// TIA Portal V20 export
FUNCTION "06 T5 EXCENTRIC Output" : Void   // FC1618, LAD
TITLE = OUTPUT
{ S7_Optimized_Access := 'TRUE' }
// stored: AutoNumber false, SetENOAutomatically false
   VAR_TEMP
      Aux_real : Real;
      Aux_dint : DInt;
      Aux_uint : UInt;
      Aux_Bool : Bool;
      Aux_OS : Bool;
   END_VAR
   VAR_TEMP   // added for the SCL form of the ladder/FBD networks
      _w1 : Bool;
      _w2 : Bool;
   END_VAR
BEGIN

REGION Network 1: ============= INTERLOCKS MOVING FORWARD =============
END_REGION

REGION Network 2: Interlocks Move FORWARD - Permanent Conditions
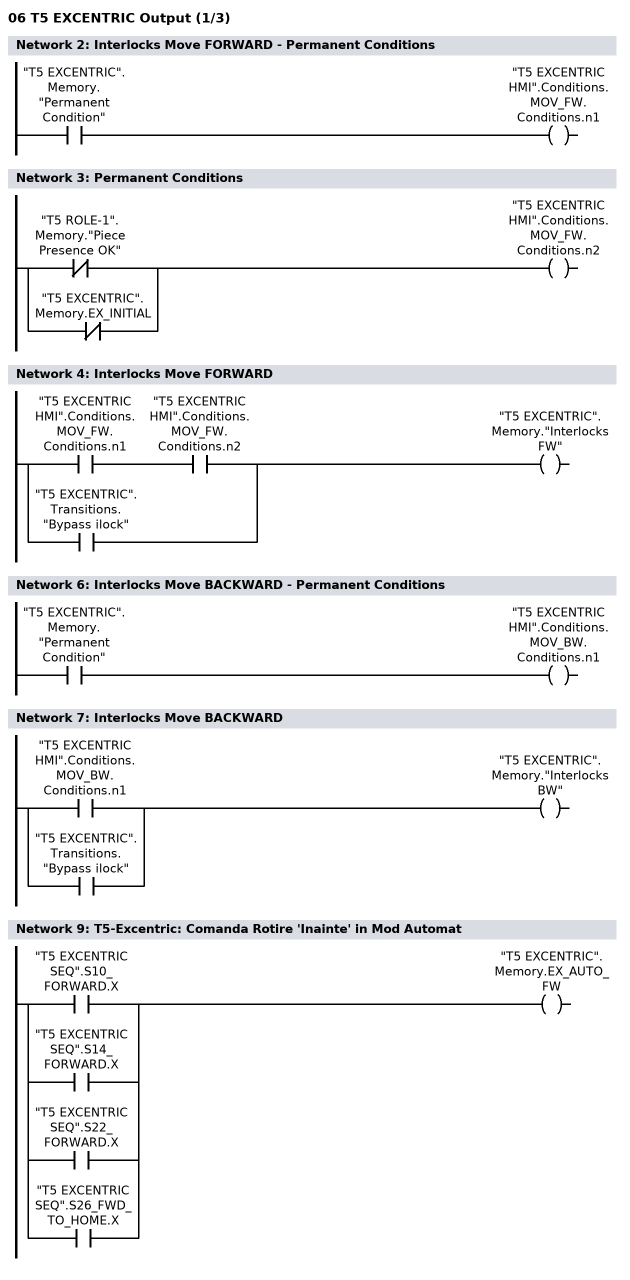
   RUNG wire#powerrail
      Contact( "T5 EXCENTRIC".Memory."Permanent Condition" )
      Coil( "T5 EXCENTRIC HMI".Conditions.MOV_FW.Conditions.n1 )
   END_RUNG
   // the same network as SCL:
   "T5 EXCENTRIC HMI".Conditions.MOV_FW.Conditions.n1 := "T5 EXCENTRIC".Memory."Permanent Condition";
END_REGION

REGION Network 3: Permanent Conditions
   RUNG wire#powerrail
      I_Contact( "T5 ROLE-1".Memory."Piece Presence OK" )
      wire#w1
      Coil( "T5 EXCENTRIC HMI".Conditions.MOV_FW.Conditions.n2 )
   END_RUNG
   RUNG wire#powerrail
      I_Contact( "T5 EXCENTRIC".Memory.EX_INITIAL )
   END_RUNG wire#w1
   // the same network as SCL:
   "T5 EXCENTRIC HMI".Conditions.MOV_FW.Conditions.n2 := NOT "T5 ROLE-1".Memory."Piece Presence OK" OR NOT "T5 EXCENTRIC".Memory.EX_INITIAL;
END_REGION

REGION Network 4: Interlocks Move FORWARD
   RUNG wire#powerrail
      Contact( "T5 EXCENTRIC HMI".Conditions.MOV_FW.Conditions.n1 )
      Contact( "T5 EXCENTRIC HMI".Conditions.MOV_FW.Conditions.n2 )
      wire#w1
      Coil( "T5 EXCENTRIC".Memory."Interlocks FW" )
   END_RUNG
   RUNG wire#powerrail
      Contact( "T5 EXCENTRIC".Transitions."Bypass ilock" )
   END_RUNG wire#w1
   // the same network as SCL:
   "T5 EXCENTRIC".Memory."Interlocks FW" := ("T5 EXCENTRIC HMI".Conditions.MOV_FW.Conditions.n1 AND "T5 EXCENTRIC HMI".Conditions.MOV_FW.Conditions.n2) OR "T5 EXCENTRIC".Transitions."Bypass ilock";
END_REGION

REGION Network 5: ============= INTERLOCKS MOVING BACKWARD =============
END_REGION

REGION Network 6: Interlocks Move BACKWARD - Permanent Conditions
   RUNG wire#powerrail
      Contact( "T5 EXCENTRIC".Memory."Permanent Condition" )
      Coil( "T5 EXCENTRIC HMI".Conditions.MOV_BW.Conditions.n1 )
   END_RUNG
   // the same network as SCL:
   "T5 EXCENTRIC HMI".Conditions.MOV_BW.Conditions.n1 := "T5 EXCENTRIC".Memory."Permanent Condition";
END_REGION

REGION Network 7: Interlocks Move BACKWARD
   RUNG wire#powerrail
      Contact( "T5 EXCENTRIC HMI".Conditions.MOV_BW.Conditions.n1 )
      wire#w1
      Coil( "T5 EXCENTRIC".Memory."Interlocks BW" )
   END_RUNG
   RUNG wire#powerrail
      Contact( "T5 EXCENTRIC".Transitions."Bypass ilock" )
   END_RUNG wire#w1
   // the same network as SCL:
   "T5 EXCENTRIC".Memory."Interlocks BW" := "T5 EXCENTRIC HMI".Conditions.MOV_BW.Conditions.n1 OR "T5 EXCENTRIC".Transitions."Bypass ilock";
END_REGION

REGION Network 8: ============ COMMANDS ============
END_REGION

REGION Network 9: T5-Excentric: Comanda Rotire 'Inainte' in Mod Automat
   RUNG wire#powerrail
      Contact( "T5 EXCENTRIC SEQ".S10_FORWARD.X )
      wire#w1
      Coil( "T5 EXCENTRIC".Memory.EX_AUTO_FW )
   END_RUNG
   RUNG wire#powerrail
      Contact( "T5 EXCENTRIC SEQ".S14_FORWARD.X )
   END_RUNG wire#w1
   RUNG wire#powerrail
      Contact( "T5 EXCENTRIC SEQ".S22_FORWARD.X )
   END_RUNG wire#w1
   RUNG wire#powerrail
      Contact( "T5 EXCENTRIC SEQ".S26_FWD_TO_HOME.X )
   END_RUNG wire#w1
   // the same network as SCL:
   "T5 EXCENTRIC".Memory.EX_AUTO_FW := "T5 EXCENTRIC SEQ".S10_FORWARD.X OR "T5 EXCENTRIC SEQ".S14_FORWARD.X OR "T5 EXCENTRIC SEQ".S22_FORWARD.X OR "T5 EXCENTRIC SEQ".S26_FWD_TO_HOME.X;
END_REGION

REGION Network 10: T5-Excentric: Comanda Rotire 'Inainte' in Mod Manual
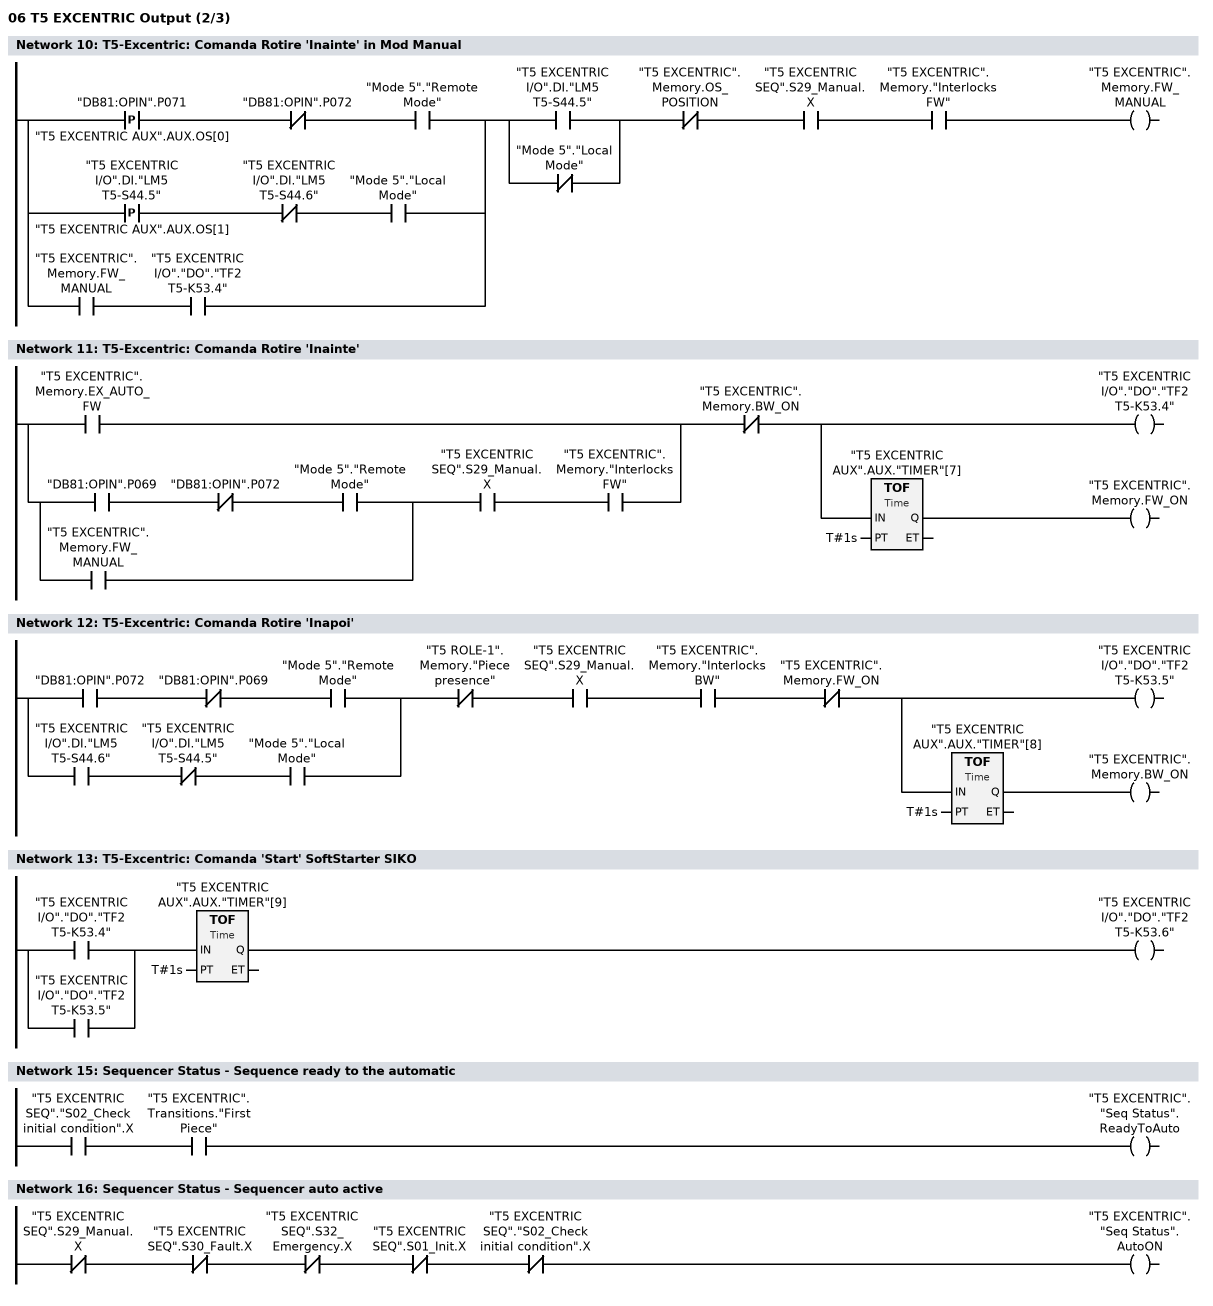
   RUNG wire#powerrail
      P_Contact(operand := "DB81:OPIN".P071, bit := "T5 EXCENTRIC AUX".AUX.OS[0])
      I_Contact( "DB81:OPIN".P072 )
      Contact( "Mode 5"."Remote Mode" )
      wire#w1
      Contact( "T5 EXCENTRIC I/O".DI."LM5 T5-S44.5" )
      wire#w2
      I_Contact( "T5 EXCENTRIC".Memory.OS_POSITION )
      Contact( "T5 EXCENTRIC SEQ".S29_Manual.X )
      Contact( "T5 EXCENTRIC".Memory."Interlocks FW" )
      Coil( "T5 EXCENTRIC".Memory.FW_MANUAL )
   END_RUNG
   RUNG wire#powerrail
      P_Contact(operand := "T5 EXCENTRIC I/O".DI."LM5 T5-S44.5", bit := "T5 EXCENTRIC AUX".AUX.OS[1])
      I_Contact( "T5 EXCENTRIC I/O".DI."LM5 T5-S44.6" )
      Contact( "Mode 5"."Local Mode" )
   END_RUNG wire#w1
   RUNG wire#powerrail
      Contact( "T5 EXCENTRIC".Memory.FW_MANUAL )
      Contact( "T5 EXCENTRIC I/O"."DO"."TF2 T5-K53.4" )
   END_RUNG wire#w1
   RUNG wire#w1
      I_Contact( "Mode 5"."Local Mode" )
   END_RUNG wire#w2
   // the same network as SCL:
   #_w1 := "DB81:OPIN".P071 AND NOT "T5 EXCENTRIC AUX".AUX.OS[0];   // rising edge of "DB81:OPIN".P071
   "T5 EXCENTRIC AUX".AUX.OS[0] := "DB81:OPIN".P071;
   #_w2 := "T5 EXCENTRIC I/O".DI."LM5 T5-S44.5" AND NOT "T5 EXCENTRIC AUX".AUX.OS[1];   // rising edge of "T5 EXCENTRIC I/O".DI."LM5 T5-S44.5"
   "T5 EXCENTRIC AUX".AUX.OS[1] := "T5 EXCENTRIC I/O".DI."LM5 T5-S44.5";
   "T5 EXCENTRIC".Memory.FW_MANUAL := ((#_w1 AND NOT "DB81:OPIN".P072 AND "Mode 5"."Remote Mode") OR (#_w2 AND NOT "T5 EXCENTRIC I/O".DI."LM5 T5-S44.6" AND "Mode 5"."Local Mode") OR ("T5 EXCENTRIC".Memory.FW_MANUAL AND "T5 EXCENTRIC I/O"."DO"."TF2 T5-K53.4")) AND ("T5 EXCENTRIC I/O".DI."LM5 T5-S44.5" OR NOT "Mode 5"."Local Mode") AND NOT "T5 EXCENTRIC".Memory.OS_POSITION AND "T5 EXCENTRIC SEQ".S29_Manual.X AND "T5 EXCENTRIC".Memory."Interlocks FW";
END_REGION

REGION Network 11: T5-Excentric: Comanda Rotire 'Inainte'
   RUNG wire#powerrail
      Contact( "T5 EXCENTRIC".Memory.EX_AUTO_FW )
      wire#w1
      I_Contact( "T5 EXCENTRIC".Memory.BW_ON )
      wire#w3
      Coil( "T5 EXCENTRIC I/O"."DO"."TF2 T5-K53.4" )
   END_RUNG
   RUNG wire#powerrail
      Contact( "DB81:OPIN".P069 )
      I_Contact( "DB81:OPIN".P072 )
      Contact( "Mode 5"."Remote Mode" )
      wire#w2
      Contact( "T5 EXCENTRIC SEQ".S29_Manual.X )
      Contact( "T5 EXCENTRIC".Memory."Interlocks FW" )
   END_RUNG wire#w1
   RUNG wire#powerrail
      Contact( "T5 EXCENTRIC".Memory.FW_MANUAL )
   END_RUNG wire#w2
   RUNG wire#w3
      { S7_Templates := "time_type := Time" } "T5 EXCENTRIC AUX".AUX."TIMER"[7].TOF(pt := T#1s, et =>)
      Coil( "T5 EXCENTRIC".Memory.FW_ON )
   END_RUNG
   // the same network as SCL:
   "T5 EXCENTRIC I/O"."DO"."TF2 T5-K53.4" := ("T5 EXCENTRIC".Memory.EX_AUTO_FW OR ((("DB81:OPIN".P069 AND NOT "DB81:OPIN".P072 AND "Mode 5"."Remote Mode") OR "T5 EXCENTRIC".Memory.FW_MANUAL) AND "T5 EXCENTRIC SEQ".S29_Manual.X AND "T5 EXCENTRIC".Memory."Interlocks FW")) AND NOT "T5 EXCENTRIC".Memory.BW_ON;
   "T5 EXCENTRIC AUX".AUX."TIMER"[7].TOF(IN := "T5 EXCENTRIC I/O"."DO"."TF2 T5-K53.4", PT := T#1s);
   "T5 EXCENTRIC".Memory.FW_ON := "T5 EXCENTRIC AUX".AUX."TIMER"[7].Q;
END_REGION

REGION Network 12: T5-Excentric: Comanda Rotire 'Inapoi'
   RUNG wire#powerrail
      Contact( "DB81:OPIN".P072 )
      I_Contact( "DB81:OPIN".P069 )
      Contact( "Mode 5"."Remote Mode" )
      wire#w1
      I_Contact( "T5 ROLE-1".Memory."Piece presence" )
      Contact( "T5 EXCENTRIC SEQ".S29_Manual.X )
      Contact( "T5 EXCENTRIC".Memory."Interlocks BW" )
      I_Contact( "T5 EXCENTRIC".Memory.FW_ON )
      wire#w2
      Coil( "T5 EXCENTRIC I/O"."DO"."TF2 T5-K53.5" )
   END_RUNG
   RUNG wire#powerrail
      Contact( "T5 EXCENTRIC I/O".DI."LM5 T5-S44.6" )
      I_Contact( "T5 EXCENTRIC I/O".DI."LM5 T5-S44.5" )
      Contact( "Mode 5"."Local Mode" )
   END_RUNG wire#w1
   RUNG wire#w2
      { S7_Templates := "time_type := Time" } "T5 EXCENTRIC AUX".AUX."TIMER"[8].TOF(pt := T#1s, et =>)
      Coil( "T5 EXCENTRIC".Memory.BW_ON )
   END_RUNG
   // the same network as SCL:
   "T5 EXCENTRIC I/O"."DO"."TF2 T5-K53.5" := (("DB81:OPIN".P072 AND NOT "DB81:OPIN".P069 AND "Mode 5"."Remote Mode") OR ("T5 EXCENTRIC I/O".DI."LM5 T5-S44.6" AND NOT "T5 EXCENTRIC I/O".DI."LM5 T5-S44.5" AND "Mode 5"."Local Mode")) AND NOT "T5 ROLE-1".Memory."Piece presence" AND "T5 EXCENTRIC SEQ".S29_Manual.X AND "T5 EXCENTRIC".Memory."Interlocks BW" AND NOT "T5 EXCENTRIC".Memory.FW_ON;
   "T5 EXCENTRIC AUX".AUX."TIMER"[8].TOF(IN := "T5 EXCENTRIC I/O"."DO"."TF2 T5-K53.5", PT := T#1s);
   "T5 EXCENTRIC".Memory.BW_ON := "T5 EXCENTRIC AUX".AUX."TIMER"[8].Q;
END_REGION

REGION Network 13: T5-Excentric: Comanda 'Start' SoftStarter SIKO
   RUNG wire#powerrail
      Contact( "T5 EXCENTRIC I/O"."DO"."TF2 T5-K53.4" )
      wire#w1
      { S7_Templates := "time_type := Time" } "T5 EXCENTRIC AUX".AUX."TIMER"[9].TOF(pt := T#1s, et =>)
      Coil( "T5 EXCENTRIC I/O"."DO"."TF2 T5-K53.6" )
   END_RUNG
   RUNG wire#powerrail
      Contact( "T5 EXCENTRIC I/O"."DO"."TF2 T5-K53.5" )
   END_RUNG wire#w1
   // the same network as SCL:
   "T5 EXCENTRIC AUX".AUX."TIMER"[9].TOF(IN := "T5 EXCENTRIC I/O"."DO"."TF2 T5-K53.4" OR "T5 EXCENTRIC I/O"."DO"."TF2 T5-K53.5",
                           PT := T#1s);
   "T5 EXCENTRIC I/O"."DO"."TF2 T5-K53.6" := "T5 EXCENTRIC AUX".AUX."TIMER"[9].Q;
END_REGION

REGION Network 14: ================== SEQUENCER STATUS ==================
END_REGION

REGION Network 15: Sequencer Status - Sequence ready to the automatic
   RUNG wire#powerrail
      Contact( "T5 EXCENTRIC SEQ"."S02_Check initial condition".X )
      Contact( "T5 EXCENTRIC".Transitions."First Piece" )
      Coil( "T5 EXCENTRIC"."Seq Status".ReadyToAuto )
   END_RUNG
   // the same network as SCL:
   "T5 EXCENTRIC"."Seq Status".ReadyToAuto := "T5 EXCENTRIC SEQ"."S02_Check initial condition".X AND "T5 EXCENTRIC".Transitions."First Piece";
END_REGION

REGION Network 16: Sequencer Status - Sequencer auto active
   RUNG wire#powerrail
      I_Contact( "T5 EXCENTRIC SEQ".S29_Manual.X )
      I_Contact( "T5 EXCENTRIC SEQ".S30_Fault.X )
      I_Contact( "T5 EXCENTRIC SEQ".S32_Emergency.X )
      I_Contact( "T5 EXCENTRIC SEQ".S01_Init.X )
      I_Contact( "T5 EXCENTRIC SEQ"."S02_Check initial condition".X )
      Coil( "T5 EXCENTRIC"."Seq Status".AutoON )
   END_RUNG
   // the same network as SCL:
   "T5 EXCENTRIC"."Seq Status".AutoON := NOT "T5 EXCENTRIC SEQ".S29_Manual.X AND NOT "T5 EXCENTRIC SEQ".S30_Fault.X AND NOT "T5 EXCENTRIC SEQ".S32_Emergency.X AND NOT "T5 EXCENTRIC SEQ".S01_Init.X AND NOT "T5 EXCENTRIC SEQ"."S02_Check initial condition".X;
END_REGION

REGION Network 17: Sequencer Status - Sequencer wait piece
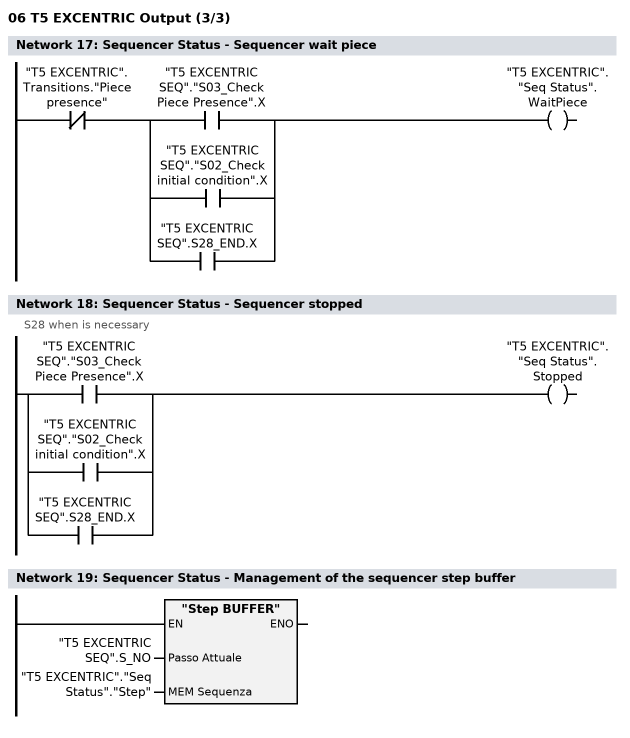
   RUNG wire#powerrail
      I_Contact( "T5 EXCENTRIC".Transitions."Piece presence" )
      wire#w1
      Contact( "T5 EXCENTRIC SEQ"."S03_Check Piece Presence".X )
      wire#w2
      Coil( "T5 EXCENTRIC"."Seq Status".WaitPiece )
   END_RUNG
   RUNG wire#w1
      Contact( "T5 EXCENTRIC SEQ"."S02_Check initial condition".X )
   END_RUNG wire#w2
   RUNG wire#w1
      Contact( "T5 EXCENTRIC SEQ".S28_END.X )
   END_RUNG wire#w2
   // the same network as SCL:
   "T5 EXCENTRIC"."Seq Status".WaitPiece := NOT "T5 EXCENTRIC".Transitions."Piece presence" AND ("T5 EXCENTRIC SEQ"."S03_Check Piece Presence".X OR "T5 EXCENTRIC SEQ"."S02_Check initial condition".X OR "T5 EXCENTRIC SEQ".S28_END.X);
END_REGION

REGION Network 18: Sequencer Status - Sequencer stopped
   // S28 when is necessary
   RUNG wire#powerrail
      Contact( "T5 EXCENTRIC SEQ"."S03_Check Piece Presence".X )
      wire#w1
      Coil( "T5 EXCENTRIC"."Seq Status".Stopped )
   END_RUNG
   RUNG wire#powerrail
      Contact( "T5 EXCENTRIC SEQ"."S02_Check initial condition".X )
   END_RUNG wire#w1
   RUNG wire#powerrail
      Contact( "T5 EXCENTRIC SEQ".S28_END.X )
   END_RUNG wire#w1
   // the same network as SCL:
   "T5 EXCENTRIC"."Seq Status".Stopped := "T5 EXCENTRIC SEQ"."S03_Check Piece Presence".X OR "T5 EXCENTRIC SEQ"."S02_Check initial condition".X OR "T5 EXCENTRIC SEQ".S28_END.X;
END_REGION

REGION Network 19: Sequencer Status - Management of the sequencer step buffer
   RUNG wire#powerrail
      "Step BUFFER"("Passo Attuale" := "T5 EXCENTRIC SEQ".S_NO, "MEM Sequenza" := "T5 EXCENTRIC"."Seq Status"."Step")
   END_RUNG
   // the same network as SCL:
   "Step BUFFER"("Passo Attuale" := "T5 EXCENTRIC SEQ".S_NO,
                 "MEM Sequenza" := "T5 EXCENTRIC"."Seq Status"."Step");
END_REGION
END_FUNCTION
